(* IEC 61131-3 sources: statemachine/src/StateFramework/State, 13 files *)

(* ---- StateControllerStatus.st ---- *)
NAMESPACE Simatic.Ax.StateFramework
    // Status and error codes reported by the state controller.
    TYPE
        StateControllerStatus : WORD (
            STATUS_NO_ERR := WORD#16#7000,
            STATUS_IS_RUNNING := WORD#16#7001,
            STATUS_STATE_CHANGED := WORD#16#7002,
            STATUS_NO_INITIALSTATE := WORD#16#8100,
            STATUS_NO_NEXTSTATE := WORD#16#8101,
            STATUS_NO_TRANSITION := WORD#16#8102
        ) := STATUS_NO_ERR;
    END_TYPE
END_NAMESPACE

(* ---- StateLogger.st ---- *)
NAMESPACE Simatic.Ax.StateFramework
    CLASS StateLogger IMPLEMENTS ILogger
        VAR PUBLIC
            // Public ring buffer that stores the most recent log messages.
            MsgBuffer : Array[0..BUF_SIZE - 1] OF LogMessage;
        END_VAR
        VAR PROTECTED

        END_VAR
        VAR PRIVATE
            // Write position inside the ring buffer.
            _pos : INT;
        END_VAR
        VAR CONSTANT PRIVATE
            // Maximum number of log entries kept in memory.
            BUF_SIZE : INT := 100;
        END_VAR

        METHOD PUBLIC WriteLog
            VAR_INPUT
                message : STRING;
            END_VAR
            VAR_TEMP
                _data : REF_TO LogMessage;
                _timestamp : DATE_AND_TIME;
            END_VAR
            // The current slot is overwritten and the write position advances circularly.
            _data := REF(MsgBuffer[_pos]);
            _data^.message := message;
            _data^.timestamp := _timestamp;
            _pos := (_pos + 1) MOD BUF_SIZE;
        END_METHOD

    END_CLASS

    TYPE
        // One buffered log entry with payload and timestamp field.
        LogMessage : STRUCT
            timestamp : DATE_AND_TIME;
            message : STRING;
        END_STRUCT;
    END_TYPE

END_NAMESPACE

(* ---- StateStatus.st ---- *)
NAMESPACE Simatic.Ax.StateFramework
    // Runtime status of a state instance inside the controller.
    TYPE
        StateStatus : (
            IDLE,
            ACTIVE
        ) := IDLE;
    END_TYPE
END_NAMESPACE

(* ---- ILogger.st ---- *)
NAMESPACE Simatic.Ax.StateFramework
    INTERFACE ILogger

        // Writes one log message to the attached logger implementation.
        METHOD WriteLog
            VAR_INPUT
                message : String;
            END_VAR
        END_METHOD
    END_INTERFACE
END_NAMESPACE

(* ---- IState.st ---- *)
NAMESPACE Simatic.Ax.StateFramework
    INTERFACE IState

        // Called once when the controller activates the state.
        METHOD OnEntry
        END_METHOD

        // Called once before the controller leaves the state.
        METHOD OnExit
        END_METHOD

        // Called in each execution cycle while the state remains active.
        METHOD Action
        END_METHOD

        // Returns the transition at the requested zero-based position.
        METHOD GetTransition : ITransition
            VAR_INPUT
                pos : UINT;
            END_VAR
        END_METHOD

        // Returns how many outgoing transitions are currently configured.
        METHOD TransitionCount : UINT
        END_METHOD

        // Returns the numeric identifier of the state.
        METHOD GetStateID : INT
        END_METHOD

        // Returns the display name of the state.
        METHOD GetStateName : STRING
        END_METHOD

        // Returns the current runtime status of the state.
        METHOD GetStatus : StateStatus
        END_METHOD

    END_INTERFACE
END_NAMESPACE

(* ---- IStateController.st ---- *)
NAMESPACE Simatic.Ax.StateFramework
    // Marker interface for state controller implementations.
    INTERFACE IStateController
    END_INTERFACE
END_NAMESPACE

(* ---- IStateMuteable.st ---- *)
NAMESPACE Simatic.Ax.StateFramework
    INTERFACE IStateMuteable

        // Allows the controller to update the runtime status of a state.
        METHOD SetStatus
            VAR_INPUT
                status : StateStatus;
            END_VAR
        END_METHOD

    END_INTERFACE
END_NAMESPACE

(* ---- AbstractState.st ---- *)
NAMESPACE Simatic.Ax.StateFramework
    CLASS ABSTRACT AbstractState IMPLEMENTS IState, IStateMuteable

        VAR PUBLIC
            Transition1 : ITransition;
            StateID : INT;
            StateName : String;
        END_VAR

        VAR PROTECTED
             _actualStatus : StateStatus;
        END_VAR

        METHOD PUBLIC ABSTRACT OnEntry
        END_METHOD

        METHOD PUBLIC ABSTRACT OnExit
        END_METHOD

        METHOD PUBLIC ABSTRACT Action
        END_METHOD

        METHOD PUBLIC GetTransition : ITransition
            VAR_INPUT
                pos : UINT;
            END_VAR
            // The base implementation supports exactly one outgoing transition.
            IF (THIS.TransitionCount() = pos + UINT#1) THEN
                GetTransition := transition1;
            ELSE
                GetTransition := NULL;
            END_IF;
        END_METHOD

        METHOD PUBLIC TransitionCount : UINT
            // A state either exposes its single configured transition or none.
            IF (transition1 <> NULL) THEN
                TransitionCount := UINT#1;
            ELSE
                TransitionCount := UINT#0;
            END_IF;
        END_METHOD

        METHOD PUBLIC GetStateID : INT
            GetStateID := StateID;
        END_METHOD

        METHOD PUBLIC FINAL GetStateName : STRING
            GetStateName := StateName;
        END_METHOD

        METHOD PUBLIC FINAL GetStatus : StateStatus
            GetStatus := _actualStatus;
        END_METHOD

        METHOD PUBLIC FINAL SetStatus
            VAR_INPUT
                status : StateStatus;
            END_VAR
            _actualStatus := status;
        END_METHOD
    END_CLASS
END_NAMESPACE

(* ---- State1Transition.st ---- *)
USING Simatic.Ax.Stateframework;

NAMESPACE Simatic.Ax.StateFramework
    // Convenience base state for exactly one outgoing transition.
    CLASS State1Transition EXTENDS AbstractState

        METHOD PUBLIC OVERRIDE OnEntry
            // Test helper state with no custom entry behavior.
            ;
        END_METHOD

        METHOD PUBLIC OVERRIDE OnExit
            // Test helper state with no custom exit behavior.
            ;
        END_METHOD

        METHOD PUBLIC OVERRIDE Action
            // Test helper state with no custom action behavior.
            ;
        END_METHOD

    END_CLASS

END_NAMESPACE

(* ---- State2Transition.st ---- *)
USING Simatic.Ax.Stateframework;

NAMESPACE Simatic.Ax.StateFramework

    // Convenience base state for up to two outgoing transitions.
    CLASS State2Transition EXTENDS AbstractState

        VAR PUBLIC
            // Optional second outgoing transition.
            Transition2 : ITransition;
        END_VAR

        METHOD PUBLIC OVERRIDE OnEntry
            // Default implementation intentionally does nothing.
            ;
        END_METHOD

        METHOD PUBLIC OVERRIDE OnExit
            // Default implementation intentionally does nothing.
            ;
        END_METHOD

        METHOD PUBLIC OVERRIDE Action
            // Default implementation intentionally does nothing.
            ;
        END_METHOD

        METHOD PUBLIC FINAL OVERRIDE GetTransition : ITransition
            VAR_INPUT
                pos : UINT;
            END_VAR
            VAR_TEMP
                cnt : UINT;
            END_VAR;

            cnt := THIS.TransitionCount();

            IF (pos >= cnt) THEN
                GetTransition := NULL;
                RETURN;
            END_IF;

            // With only one configured transition, the populated slot is returned as index 0.
            IF (cnt = UINT#1) THEN
                IF (transition1 <> NULL) THEN
                    GetTransition := transition1;
                ELSE
                    GetTransition := transition2;
                END_IF;
            ELSE
                CASE pos OF
                    UINT#0: GetTransition := transition1;
                    UINT#1: GetTransition := transition2;
                ELSE
                    GetTransition := NULL;
                END_CASE;
            END_IF;

        END_METHOD

        METHOD PUBLIC FINAL OVERRIDE TransitionCount : UINT
            // Counts how many of the two transition slots are populated.
            IF (transition1 = NULL AND transition2 = NULL) THEN
                TransitionCount := UINT#0;
            ELSIF (transition1 <> NULL AND transition2 <> NULL) THEN
                TransitionCount := UINT#2;
            ELSE
                TransitionCount := UINT#1;
            END_IF;
        END_METHOD
    END_CLASS

END_NAMESPACE

(* ---- State3Transition.st ---- *)
USING Simatic.Ax.Stateframework;

NAMESPACE Simatic.Ax.StateFramework

    // Convenience base state for up to three outgoing transitions.
    CLASS State3Transition EXTENDS AbstractState

        VAR PUBLIC
            // Optional second outgoing transition.
            Transition2 : ITransition;
            // Optional third outgoing transition.
            Transition3 : ITransition;
        END_VAR

        METHOD PUBLIC OVERRIDE OnEntry
            // Default implementation intentionally does nothing.
            ;
        END_METHOD

        METHOD PUBLIC OVERRIDE OnExit
            // Default implementation intentionally does nothing.
            ;
        END_METHOD

        METHOD PUBLIC OVERRIDE Action
            // Default implementation intentionally does nothing.
            ;
        END_METHOD

        METHOD PUBLIC FINAL OVERRIDE GetTransition : ITransition
            VAR_INPUT
                pos : UINT;
            END_VAR
            VAR_TEMP
                cnt : UINT;
            END_VAR;

            cnt := THIS.TransitionCount();

            IF (pos >= cnt) THEN
                GetTransition := NULL;
                RETURN;
            END_IF;

            // With only one configured transition, the populated slot is returned as index 0.
            IF (cnt = UINT#1) THEN
                IF (transition1 <> NULL) THEN
                    GetTransition := transition1;
                ELSIF (transition2 <> NULL) THEN
                    GetTransition := transition2;
                ELSE
                    GetTransition := transition3;
                END_IF;
            ELSE
                CASE pos OF
                    UINT#0: GetTransition := transition1;
                    UINT#1: GetTransition := transition2;
                    UINT#2: GetTransition := transition3;
                ELSE
                    GetTransition := NULL;
                END_CASE;
            END_IF;

        END_METHOD

        METHOD PUBLIC FINAL OVERRIDE TransitionCount : UINT
            // Counts how many of the three transition slots are populated.
            IF (transition1 = NULL AND transition2 = NULL AND transition3 = NULL) THEN
                TransitionCount := UINT#0;
            ELSIF (transition1 <> NULL AND transition2 <> NULL AND transition3 <> NULL) THEN
                TransitionCount := UINT#3;
            ELSIF (transition1 <> NULL AND transition2 <> NULL AND transition3 = NULL) THEN
                TransitionCount := UINT#2;
            ELSIF (transition1 <> NULL AND transition2 = NULL AND transition3 <> NULL) THEN
                TransitionCount := UINT#2;
            ELSIF (transition1 = NULL AND transition2 <> NULL AND transition3 <> NULL) THEN
                TransitionCount := UINT#2;
            ELSE
                TransitionCount := UINT#1;
            END_IF;
        END_METHOD
    END_CLASS

END_NAMESPACE

(* ---- StateController.st ---- *)
NAMESPACE Simatic.Ax.StateFramework
    CLASS StateController IMPLEMENTS IStateController

        VAR PUBLIC
            InitialState: IState;
            Logger : ILogger;
        END_VAR

        VAR PRIVATE
            _status : StateControllerStatus;
            _statesActive : INT;
        END_VAR

        VAR PROTECTED
            _activeStateId : INT;
            _activeStateName : String;
            _lastState : INT;
            _activeState : IState;
        END_VAR

        METHOD PUBLIC FINAL Execute
            VAR_TEMP
                states : INT;
            END_VAR

            // The controller cannot start without a configured entry state.
            IF (InitialState = NULL) THEN
                _status := StateControllerStatus#STATUS_NO_INITIALSTATE;
                RETURN;
            END_IF;

            // Error states are latched and block further execution cycles.
            IF (THIS.HasError()) THEN
                RETURN;
            END_IF;

            // The first cycle activates the initial state before evaluating transitions.
            IF (_activeState = NULL) THEN
                THIS.ActivateState(InitialState);
            END_IF;

            _statesActive := 1;
            THIS.ExecuteState(_activeState);

        END_METHOD

        /// Terminates the actual state and start with the InitialState
        METHOD PUBLIC Restart : IState
            // Restart terminates the current state and re-enters the configured initial state.
            IF (_activeState <> NULL) THEN
                THIS.TerminateState(_activeState);
            END_IF;
            IF (InitialState <> NULL) THEN
                THIS.ActivateState(InitialState);
                Restart := InitialState;
            ELSE
                Restart := NULL;
            END_IF;

        END_METHOD

        /// Terminates state
        /// Call the OnExit method of the actual state
        /// Reset all guards
        METHOD PRIVATE TerminateState
            VAR_INPUT
                state : IState;
            END_VAR
            VAR_TEMP
                _muetabaleState : IStateMuteable;
            END_VAR
            state.OnExit();
            _lastState := state.GetStateId();

            // Reset guards of the state that is being left so counters and timers start fresh.
            THIS.ResetGuards();

            // Mutable states are marked idle after OnExit has completed.
            _muetabaleState ?= state;
            IF (_muetabaleState <> NULL) THEN
                _muetabaleState.SetStatus(status := StateStatus#Idle);
            END_IF;
        END_METHOD

        METHOD PRIVATE ActivateState
            VAR_INPUT
                state : IState;
            END_VAR
            VAR_TEMP
                _muetabaleState : IStateMuteable;
            END_VAR
            _activeState := state;
            _status := StateControllerStatus#STATUS_STATE_CHANGED;
            _activeStateId := _activeState.GetStateId();
            _activeStateName := _activeState.GetStateName();
            // Mutable states are marked active before OnEntry is called.
            _muetabaleState ?= state;
            IF (_muetabaleState <> NULL) THEN
                _muetabaleState.SetStatus(status := StateStatus#Active);
            END_IF;

            // OnEntry is called exactly once per activation after the controller has marked the state active.
            _activeState.OnEntry();
        END_METHOD

        METHOD PRIVATE ExecuteState
            VAR_INPUT
                activeState : IState;
            END_VAR
            VAR_TEMP
                transition : UINT;
                actualTransition : ITransition;
                actualGuard : IGuard;
                nextState : IState;
            END_VAR

            IF (_activeState.TransitionCount() > UINT#0) THEN
                FOR transition := UINT#0 TO _activeState.TransitionCount() - UINT#1 DO
                    actualTransition := _activeState.GetTransition(pos := transition);

                    IF (actualTransition = NULL) THEN
                        CONTINUE;
                    END_IF;

                    actualGuard := actualTransition.GetGuard();
                    IF (actualGuard = NULL) THEN
                        CONTINUE;
                    END_IF;

                    IF (actualGuard.Check()) THEN

                        // The first guard that evaluates to TRUE wins the transition.
                        THIS.TerminateState(_activeState);
                        nextState := actualTransition.GetNextState();
                        _activeState := nextState;

                        // A taken transition without a target state is treated as a configuration error.
                        IF (_activeState = NULL) THEN
                            _status := StateControllerStatus#STATUS_NO_NEXTSTATE;
                            RETURN;
                        END_IF;

                        // The new state is entered immediately and may run its Action in the same cycle.
                        THIS.ActivateState(_activeState);

                        EXIT;
                    END_IF;
                END_FOR;
            ELSE
                // States without outgoing transitions stop the controller with STATUS_NO_TRANSITION.
                _status := StateControllerStatus#STATUS_NO_TRANSITION;
                RETURN;
            END_IF;

            // Action is executed after transition evaluation on the currently active state.
            _status := StateControllerStatus#STATUS_IS_RUNNING;
            _activeState.Action();
        END_METHOD

        // Reset all guards of the active state after a successful state change.
        METHOD PRIVATE ResetGuards
            VAR_TEMP
                actualTransition : UINT;
                transitionRef : ITransition;
                guardRef : IGuard;
            END_VAR
            IF (_activeState.TransitionCount() > UINT#0) THEN
                FOR actualTransition := UINT#0 TO _activeState.TransitionCount() - UINT#1 DO
                    transitionRef := _activeState.GetTransition(pos := actualTransition);
                    IF (transitionRef = NULL) THEN
                        CONTINUE;
                    END_IF;

                    guardRef := transitionRef.GetGuard();
                    IF (guardRef <> NULL) THEN
                        guardRef.Reset();
                    END_IF;
                END_FOR;
            END_IF;
        END_METHOD

        METHOD PRIVATE HasError : BOOL
            // Error codes are encoded above 16#8000 in the status enum.
            IF (_status > WORD#16#8000) THEN
                HasError := TRUE;
            ELSE
                HasError := FALSE;
            END_IF;
        END_METHOD

        METHOD PUBLIC GetState : StateControllerStatus
            GetState := _status;
            ;
        END_METHOD

        METHOD PUBLIC GetActiveStateName : String
            GetActiveStateName := _activeStateName;
        END_METHOD

        METHOD PRIVATE LogMessage
            VAR_INPUT
                msg : String;
            END_VAR
            // Logging is optional and only forwarded when a logger implementation is attached.
            IF (Logger <> NULL) THEN
                Logger.WriteLog(msg);
            END_IF;
        END_METHOD

    END_CLASS
END_NAMESPACE

(* ---- StatemachineController.st ---- *)
NAMESPACE Simatic.Ax.StateFramework
    // Named values for states

    CLASS StatemachineController

        VAR PUBLIC
            InitialState: IState;
            Logger : ILogger;
        END_VAR

        VAR PRIVATE
            _status : StateControllerStatus;
            _statesActive : INT;
        END_VAR

        VAR PROTECTED
            _activeStateId : INT;
            _activeStateName : String;
            _lastState : INT;
            _activeState : IState;
        END_VAR

        METHOD PUBLIC FINAL Execute
            VAR_TEMP
                states : INT;
            END_VAR

            IF (InitialState = NULL) THEN
                _status := StateControllerStatus#STATUS_NO_INITIALSTATE;
                RETURN;
            END_IF;

            // dont execute if any error is active --> NULL Pointer execption
            IF (THIS.HasError()) THEN
                RETURN;
            END_IF;

            IF (_activeState = NULL) THEN
                THIS.ActivateState(InitialState);
            END_IF;

            _statesActive := 1;
            THIS.ExecuteState(_activeState);

        END_METHOD

        METHOD PRIVATE TerminateState
            VAR_INPUT
                state : IState;
            END_VAR
            ;
        END_METHOD

        METHOD PRIVATE ActivateState
            VAR_INPUT
                state : IState;
            END_VAR
            _activeState := state;
            _status := StateControllerStatus#STATUS_STATE_CHANGED;
            _activeStateId := _activeState.GetStateId();
            _activeStateName := _activeState.GetStateName();
            // Call OnEntry method of new state
            _activeState.OnEntry();
        END_METHOD

        METHOD PRIVATE ExecuteState
            VAR_INPUT
                activeState : IState;
            END_VAR
            VAR_TEMP
                transition : UINT;
                actualTransition : ITransition;
            END_VAR

            IF (_activeState.TransitionCount() > UINT#0) THEN
                FOR transition := UINT#0 TO _activeState.TransitionCount() - UINT#1 DO
                    actualTransition := _activeState.GetTransition(pos := transition);

                    IF (actualTransition = NULL) THEN
                        CONTINUE;
                    END_IF;

                    IF (actualTransition.GetGuard().Check()) THEN
                        _activeState.Action();
                        _activeState.OnExit();
                        _lastState := _activeState.GetStateId();

                        // Reset all other guards
                        THIS.ResetGuards();

                        // switchover state
                        THIS.TerminateState(_activeState);
                        // TODO write new state into list
                        _activeState := actualTransition.GetNextState();

                        // If no next state available, RETURN and set status to Error-Code --> state machine will not be executed
                        IF (_activeState = NULL) THEN
                            _status := StateControllerStatus#STATUS_NO_NEXTSTATE;
                            RETURN;
                        END_IF;

                        // Activate State
                        THIS.ActivateState(_activeState);

                        // store active state (simple state logging)
                        EXIT;
                    END_IF;
                END_FOR;
            END_IF;
            _status := StateControllerStatus#STATUS_IS_RUNNING;
            // TODO action will be called after OnExit --> has to be changed
            _activeState.Action();
        END_METHOD

        // Reset all Guards when one of the guards has Chack() = TRUE
        METHOD PRIVATE ResetGuards
            VAR_TEMP
                actualTransition : UINT;
            END_VAR
            IF (_activeState.TransitionCount() > UINT#0) THEN
                FOR actualTransition := UINT#0 TO _activeState.TransitionCount() - UINT#1 DO
                    _activeState.GetTransition(pos := actualTransition).GetGuard().Reset();
                END_FOR;
            END_IF;
        END_METHOD

        METHOD PRIVATE HasError : BOOL
            IF (_status > WORD#16#8000) THEN
                HasError := TRUE;
            ELSE
                HasError := FALSE;
            END_IF;
        END_METHOD

        METHOD PUBLIC GetState : StateControllerStatus
            GetState := _status;
            ;
        END_METHOD

        METHOD PUBLIC GetActiveStateName : String
            GetActiveStateName := _activeStateName;
        END_METHOD

        METHOD PRIVATE LogMessage
            VAR_INPUT
                msg : String;
            END_VAR
            IF (Logger <> NULL) THEN
                Logger.WriteLog(msg);
            END_IF;
        END_METHOD

    END_CLASS
END_NAMESPACE
